FUNCTION_BLOCK FB_DummyHA IMPLEMENTS I_HigherAuthority, I_LowerAuthority
VAR_INPUT
END_VAR
VAR_OUTPUT
END_VAR
VAR
END_VAR

METHOD CheckRequest : BOOL
VAR_INPUT
	nReqID	: DWORD;
END_VAR
CheckRequest := TRUE;
END_METHOD

// <Arbiter Internal>
// Elevates the arbitrated BP set to something above.
// Could be another arbiter, or a BP requester/ IO, 
// or an FB that locks in a specific portion of the BP set.
METHOD ElevateRequest : BOOL 
VAR_INPUT
    HigherAuthority : I_HigherAuthority;
END_VAR
END_METHOD

PROPERTY nLowerAuthorityID : DWORD
GET
nLowerAuthorityID := PMPS_GVL.EXCLUDED_ASSERTION_ID;
END_GET
END_PROPERTY

{warning 'add method implementation'}
METHOD RemoveRequest : BOOL
VAR_INPUT
	(*StateID to remove*)
	nReqID	: DWORD;
END_VAR
END_METHOD

{warning 'add method implementation'}
METHOD RequestBP : BOOL
VAR_INPUT
	(*StateID of state requesting beam parameter set*)
	nReqID	: DWORD;
	(*Requested beam params*)
	stReqBP	: ST_BeamParams;
END_VAR
END_METHOD

END_FUNCTION_BLOCK

(* stored: Version 1.1.0.1, ProductVersion 3.1.4022.18
   POU FB_DummyHA: Id {670c3d93-34b2-4592-94f3-5ed3a0dba153}, SpecialFunc None
   Method CheckRequest: Id {6032c3d9-45c7-4cc0-b102-000af7719efd}
   Method ElevateRequest: Id {f71f404d-56b3-451d-b2b2-c6689b13e32e}
   Property nLowerAuthorityID: Id {32132f8f-263b-4eb5-946b-8283dbd45b0c}
   Get Get: Id {e7806d6e-95f6-4d6c-bc9b-d36d07b4562a}
   Method RemoveRequest: Id {8cc18e1a-c7b1-4978-8d42-4efdc8839d77}
   Method RequestBP: Id {55d2a094-bf30-435f-a214-786bf412cbdf} *)
